FUNCTION F_GetDefaultScoringBlade : ST_SawBladeData
VAR_INPUT
END_VAR
VAR
END_VAR

F_GetDefaultScoringBlade.rBladeDiameter := 120.0;
F_GetDefaultScoringBlade.rBladeRadius := F_GetDefaultScoringBlade.rBladeDiameter / 2;
F_GetDefaultScoringBlade.rBladeThickness := 2.8;
F_GetDefaultScoringBlade.sBladeType := 'KWO split scoring saw blade';

END_FUNCTION

(* stored: Version 1.1.0.1
   POU F_GetDefaultScoringBlade: Id {63204ffb-2f62-4675-ab5e-2b993132ac0c}, SpecialFunc None *)
